// Mitsubishi GX Works2 project: kolokvijum   PLC: FX3U/FX3UC

// task Task_01 (event TRUE, interval 0, priority 31): POU_01

PROGRAM POU_01
VAR
  zona_uslova_1 : zona_uslova;
  start : BOOL;
  stopp : BOOL;
  pokreni : BOOL;
  S_1 : BOOL;
  S_2 : BOOL;
  stanje0 : BOOL;
  stanje1 : BOOL;
  stanje2 : BOOL;
  stanje3 : BOOL;
  stanje4 : BOOL;
  global_ukljuceno : BOOL;
  predji0_1 : BOOL;
  predji1_2 : BOOL;
  predji2_3 : BOOL;
  predji3_4 : BOOL;
  predji4_0 : BOOL;
  vrijeme : TIME;
  zona_prelaza_1 : zona_prelaza;
  zona_prelaza_2 : zona_prelaza;
  stanje : INT;
  zona_izlaza_1 : zona_izlaza;
  puni : BOOL;
  prazni : BOOL;
  mjesalica : BOOL;
  alarm : BOOL;
  izvrseno : BOOL;
  V_2 : BOOL;
  V_1 : BOOL;
END_VAR
(* structured ladder/FBD written out as ST: instructions are called as NAME(EN, inputs, outputs); _pN, _eN, _tN stand for wires *)
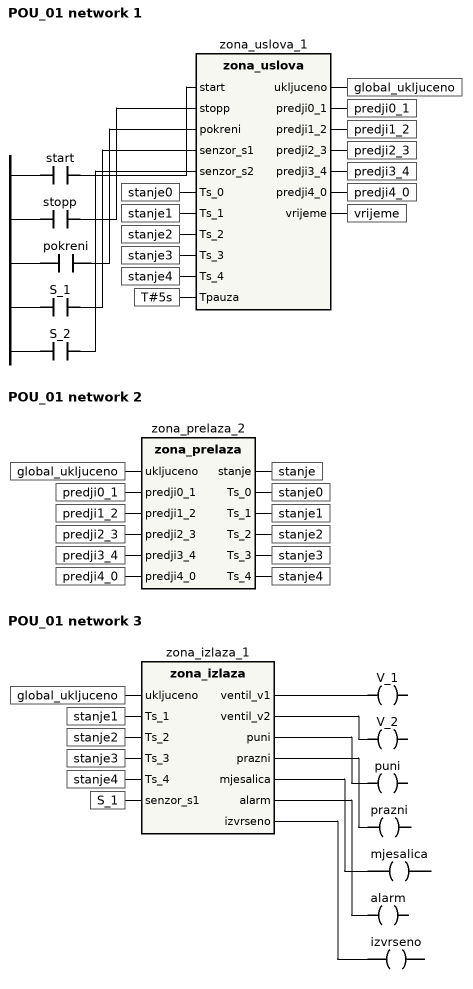
(* network 1 *)
zona_uslova_1(start := start, stopp := stopp, pokreni := pokreni, senzor_s1 := S_1, senzor_s2 := S_2, Ts_0 := stanje0, Ts_1 := stanje1, Ts_2 := stanje2, Ts_3 := stanje3, Ts_4 := stanje4, Tpauza := T#5s, ukljuceno => global_ukljuceno, predji0_1 => predji0_1, predji1_2 => predji1_2, predji2_3 => predji2_3, predji3_4 => predji3_4, predji4_0 => predji4_0, vrijeme => vrijeme);
(* network 2 *)
zona_prelaza_2(ukljuceno := global_ukljuceno, predji0_1 := predji0_1, predji1_2 := predji1_2, predji2_3 := predji2_3, predji3_4 := predji3_4, predji4_0 := predji4_0, stanje => stanje, Ts_0 => stanje0, Ts_1 => stanje1, Ts_2 => stanje2, Ts_3 => stanje3, Ts_4 => stanje4);
(* network 3 *)
zona_izlaza_1(ukljuceno := global_ukljuceno, Ts_1 := stanje1, Ts_2 := stanje2, Ts_3 := stanje3, Ts_4 := stanje4, senzor_s1 := S_1);
V_1 := zona_izlaza_1.ventil_v1;
V_2 := zona_izlaza_1.ventil_v2;
puni := zona_izlaza_1.puni;
prazni := zona_izlaza_1.prazni;
mjesalica := zona_izlaza_1.mjesalica;
alarm := zona_izlaza_1.alarm;
izvrseno := zona_izlaza_1.izvrseno;
END_PROGRAM

FUNCTION_BLOCK zona_uslova
VAR_INPUT
  start : BOOL;
  stopp : BOOL;
END_VAR
VAR_OUTPUT
  ukljuceno : BOOL;
END_VAR
VAR
  TON_1 : TON;
END_VAR
VAR_INPUT
  pokreni : BOOL;
  senzor_s1 : BOOL;
  senzor_s2 : BOOL;
  Ts_0 : BOOL;
  Ts_1 : BOOL;
  Ts_2 : BOOL;
  Ts_3 : BOOL;
  Ts_4 : BOOL;
  Tpauza : TIME;
END_VAR
VAR_OUTPUT
  predji0_1 : BOOL;
  predji1_2 : BOOL;
  predji2_3 : BOOL;
  predji3_4 : BOOL;
  predji4_0 : BOOL;
  vrijeme : TIME;
END_VAR
(* structured ladder/FBD written out as ST: instructions are called as NAME(EN, inputs, outputs); _pN, _eN, _tN stand for wires *)
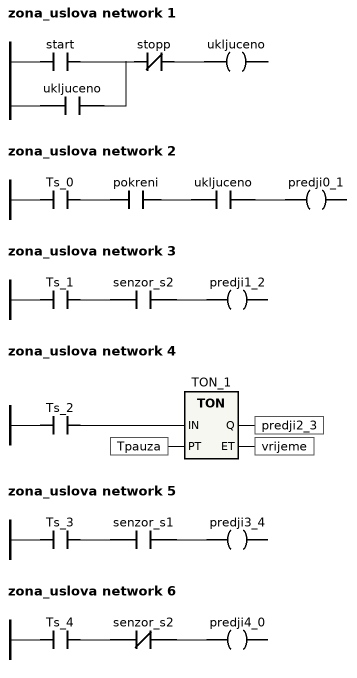
(* network 1 *)
ukljuceno := (start OR ukljuceno) AND NOT stopp;
(* network 2 *)
predji0_1 := Ts_0 AND pokreni AND ukljuceno;
(* network 3 *)
predji1_2 := Ts_1 AND senzor_s2;
(* network 4 *)
TON_1(IN := Ts_2, PT := Tpauza, Q => predji2_3, ET => vrijeme);
(* network 5 *)
predji3_4 := Ts_3 AND senzor_s1;
(* network 6 *)
predji4_0 := Ts_4 AND NOT senzor_s2;
END_FUNCTION_BLOCK

FUNCTION_BLOCK zona_prelaza
VAR_OUTPUT
  stanje : INT;
END_VAR
VAR
  jednako : ARRAY [0..2] OF BOOL;
END_VAR
VAR_INPUT
  ukljuceno : BOOL;
  predji0_1 : BOOL;
  predji1_2 : BOOL;
  predji2_3 : BOOL;
  predji3_4 : BOOL;
  predji4_0 : BOOL;
END_VAR
VAR_OUTPUT
  Ts_0 : BOOL;
  Ts_1 : BOOL;
  Ts_2 : BOOL;
  Ts_3 : BOOL;
  Ts_4 : BOOL;
END_VAR
(* structured ladder/FBD written out as ST: instructions are called as NAME(EN, inputs, outputs); _pN, _eN, _tN stand for wires *)
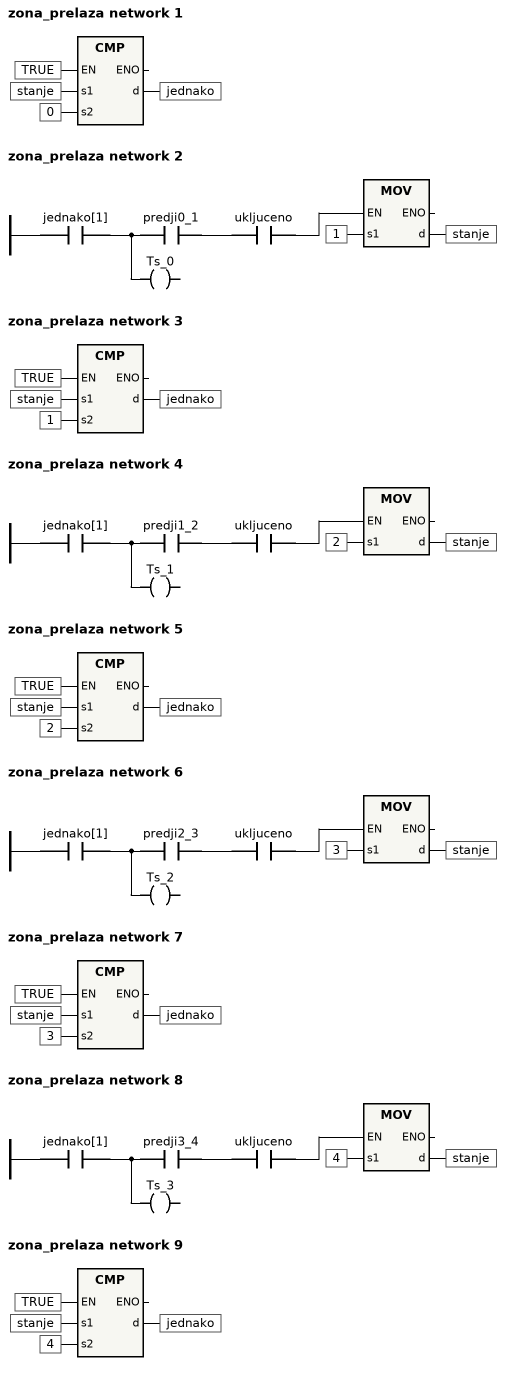
(* network 1 *)
CMP(TRUE, stanje, 0, jednako);
(* network 2 *)
MOV(jednako[1] AND predji0_1 AND ukljuceno, 1, stanje);
Ts_0 := jednako[1];
(* network 3 *)
CMP(TRUE, stanje, 1, jednako);
(* network 4 *)
MOV(jednako[1] AND predji1_2 AND ukljuceno, 2, stanje);
Ts_1 := jednako[1];
(* network 5 *)
CMP(TRUE, stanje, 2, jednako);
(* network 6 *)
MOV(jednako[1] AND predji2_3 AND ukljuceno, 3, stanje);
Ts_2 := jednako[1];
(* network 7 *)
CMP(TRUE, stanje, 3, jednako);
(* network 8 *)
MOV(jednako[1] AND predji3_4 AND ukljuceno, 4, stanje);
Ts_3 := jednako[1];
(* network 9 *)
CMP(TRUE, stanje, 4, jednako);
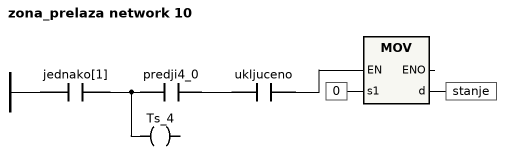
(* network 10 *)
MOV(jednako[1] AND predji4_0 AND ukljuceno, 0, stanje);
Ts_4 := jednako[1];
END_FUNCTION_BLOCK

FUNCTION_BLOCK broj_ciklusa
VAR
  broj_ciklusa : INT;
END_VAR
VAR_INPUT
  okini : BOOL;
END_VAR
VAR
  poredi : ARRAY [0..2] OF BOOL;
END_VAR
VAR_OUTPUT
  izvrseno : BOOL;
END_VAR
(* structured ladder/FBD written out as ST: instructions are called as NAME(EN, inputs, outputs); _pN, _eN, _tN stand for wires *)
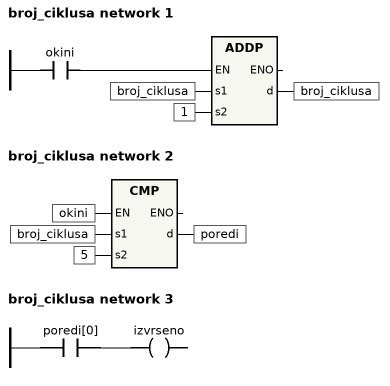
(* network 1 *)
ADDP(okini, broj_ciklusa, 1, broj_ciklusa);
(* network 2 *)
CMP(okini, broj_ciklusa, 5, poredi);
(* network 3 *)
izvrseno := poredi[0];
END_FUNCTION_BLOCK

FUNCTION_BLOCK zona_izlaza
VAR_INPUT
  ukljuceno : BOOL;
  Ts_1 : BOOL;
  Ts_2 : BOOL;
  Ts_3 : BOOL;
  Ts_4 : BOOL;
  senzor_s1 : BOOL;
END_VAR
VAR_OUTPUT
  ventil_v1 : BOOL;
  ventil_v2 : BOOL;
  puni : BOOL;
  prazni : BOOL;
  mjesalica : BOOL;
  alarm : BOOL;
  izvrseno : BOOL;
END_VAR
VAR
  broj_ciklusa_1 : broj_ciklusa;
END_VAR
(* structured ladder/FBD written out as ST: instructions are called as NAME(EN, inputs, outputs); _pN, _eN, _tN stand for wires *)
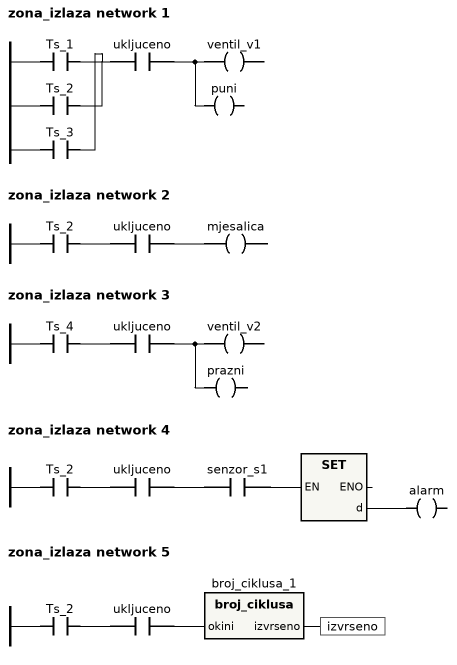
(* network 1 *)
_p1 := (Ts_1 OR Ts_2 OR Ts_3) AND ukljuceno;
ventil_v1 := _p1;
puni := _p1;
(* network 2 *)
mjesalica := Ts_2 AND ukljuceno;
(* network 3 *)
_p1 := Ts_4 AND ukljuceno;
ventil_v2 := _p1;
prazni := _p1;
(* network 4 *)
SET(Ts_2 AND ukljuceno AND senzor_s1, _t1);
alarm := _t1;
(* network 5 *)
broj_ciklusa_1(okini := Ts_2 AND ukljuceno, izvrseno => izvrseno);
END_FUNCTION_BLOCK
